PROGRAM SecondPOU
VAR
END_VAR

END_PROGRAM

(* stored: Version 1.1.0.1, ProductVersion 3.1.4026.6
   POU SecondPOU: Id {33d9a411-3250-48b9-9bf5-3199e9066c04}, SpecialFunc None *)
